FUNCTION TryConvert_BOOL_TO_UINT : BOOL
VAR_INPUT
	in : BOOL;
	out : REFERENCE TO UINT;
END_VAR

out := BOOL_TO_UINT(in);
TryConvert_BOOL_TO_UINT := TRUE;

END_FUNCTION

(* stored: Version 1.1.0.1, ProductVersion 3.1.4024.12
   POU TryConvert_BOOL_TO_UINT: Id {557b4e01-4285-4386-a7b1-e95a2dbb12ab}, SpecialFunc None *)
